TYPE UNION_oSchunkProcessData :
UNION
	Schunk_out 		: ARRAY [0..11] OF WORD;
	oSchunk_ProcessData	: oSchunkProcessData;
END_UNION
END_TYPE

(* stored: Version 1.1.0.1, ProductVersion 3.1.4024.11
   DUT UNION_oSchunkProcessData: Id {ff0b4f41-0154-4b2f-ba32-6cb429ffaa5f} *)
